(* CODESYS project Projeto_Silos.project

Project tree, tasks and I/O mapping:
  Device : CODESYS Control Win V3, 3S - Smart Software Solutions GmbH, order no. 305021, version 3.5.11.40
    application Application
      libraries: Standard, * (System)
      task Task_Simulacao (cyclic, interval t#20ms, priority 10) calls PRG_Simulacao
      task Task_Controle (cyclic, interval t#100ms, priority 5) calls PRG_Controle
      program PLC_PRG [ST]
      global variables GVL_IO
      global variables GVL_SCADA
      program PRG_Simulacao [ST]
      program PRG_Controle [SFC]: Enchimento, Acao_Parar_Tudo, Acao_Mover_SL01, Parar, Decisao_Alvo, Monitoramento_Falha, Comando_Atuadores, Adicionar_Peso, Remover_Peso
      Symbols
*)

// Device/Application/GVL_IO
VAR_GLOBAL
	
 
    (* ENTRADAS DO CLP (Sinais lidos e simulados pelo PRG_Simulacao) *)
   
    LS_01 : BOOL; (* Chave fim-de-curso Silo 1. TRUE quando Tripper posicionado. *)
    LS_02 : BOOL; (* Chave fim-de-curso Silo 2. *)
    LS_03 : BOOL; (* Chave fim-de-curso Silo 3. *)
    LS_04 : BOOL; (* Chave fim-de-curso Silo 4. *)
    
    TR_DIST : REAL; (* Sensor de distância a laser (metragem) . *)
    WT_01   : REAL; (* Balança de fluxo interna ao tripper (kg/s) . *)

 
    (* SAÍDAS DO CLP (Atuadores comandados pelo PRG_Controle) *)
  
    TR_FW   : BOOL; (* Acionamento frente do Tripper. *)
    TR_BW   : BOOL; (* Acionamento ré do Tripper. *)
    TR_VEL  : REAL; (* Velocidade de deslocamento do Tripper (m/s) . *)
    M_CT_01 : BOOL; (* Liga/desliga a correia alimentadora CT-01. *)
    BUZINA  : BOOL; (* Ativa a Buzina para sinalização. *)

END_VAR

// Device/Application/GVL_SCADA
VAR_GLOBAL
	
   
    (* COMANDOS/ENTRADAS LÓGICAS DO SCADA (Comandos para o CLP) *)

    LIGA_AUTO : BOOL; (* Comando de LIGA / DESLIGA executado via SCADA. *)
    EMG       : BOOL; (* Sinalização manual de Emergência via SCADA. *)
    REARME    : BOOL; (* Sinalização manual de Rearme via SCADA. *)
    
    FV_01     : BOOL; (* Válvula on-off de descarga Silo 1. *)
    FV_02     : BOOL; (* Válvula on-off de descarga Silo 2. *)
    FV_03     : BOOL; (* Válvula on-off de descarga Silo 3. *)
    FV_04     : BOOL; (* Válvula on-off de descarga Silo 4. *)
    
    LT_01     : REAL; (* Sensor de nível Silo 1 (Simulado manualmente via IHM, conforme orientação [cite: 123]). *)
    LT_02     : REAL; (* Sensor de nível Silo 2 (Simulado manualmente via IHM). *)
    LT_03     : REAL; (* Sensor de nível Silo 3 (Simulado manualmente via IHM). *)
    LT_04     : REAL; (* Sensor de nível Silo 4 (Simulado manualmente via IHM). *)

    
    (* DADOS/STATUS PARA VISUALIZAÇÃO NO SCADA (CLP envia para IHM) *)

    PESO_SL_01 : REAL; (* Peso total em toneladas do Silo 1[cite: 94]. *)
    PESO_SL_02 : REAL; (* Peso total em toneladas do Silo 2. *)
    PESO_SL_03 : REAL; (* Peso total em toneladas do Silo 3. *)
    PESO_SL_04 : REAL; (* Peso total em toneladas do Silo 4. *)
    
    STATUS_FALHA : BOOL; (* Indica que o CLP entrou em modo FALHA[cite: 64]. *)
    STATUS_EMG   : BOOL; (* Status da Emergência (para Alarme). *)
    POS_TRIPPER  : REAL; (* Posição atual do Tripper para Animação Visual. *)
    
    (* Variáveis para simulação de falha das chaves Fim-de-Curso via IHM [cite: 133] *)
    FALHA_LS_01 : BOOL;
    FALHA_LS_02 : BOOL;
    FALHA_LS_03 : BOOL;
    FALHA_LS_04 : BOOL;
	
	siloAlvo     : INT := 0; (* Silo alvo do tripper *)
	carregando   : BOOL;
	
END_VAR

// Device/Application/PRG_Simulacao
PROGRAM PRG_Simulacao
(* ==========================================================
 1. DECLARAÇÃO DE TODAS AS VARIÁVEIS
==========================================================
*)

(* Variáveis Temporárias *)
VAR
    fDeslocamentoCiclo : REAL;
END_VAR

(* Variáveis Constantes para posições *)
VAR CONSTANT
    fPosSilo_01 : REAL := 00.0; (* Posição central do Silo 1 em metros *)
    fPosSilo_02 : REAL := 10.0; (* Posição central do Silo 2 em metros *)
    fPosSilo_03 : REAL := 20.0; (* Posição central do Silo 3 em metros *)
    fPosSilo_04 : REAL := 30.0; (* Posição central do Silo 4 em metros *)
    fMargemPos  : REAL := 0.1;  (* Margem de 10cm para considerar "centro" *)
	fLimiteMaxPista : REAL := 30.0; (* A pista termina no silo 4 (30m)*)
END_VAR

(* ========================================================== 
 2. INÍCIO DA LÓGICA DO PROGRAMA 
==========================================================
*)

(* ==========================================================
 2.1 CÁLCULO DO DESLOCAMENTO DO TRIPPER (TR_DIST) 
==========================================================
*)
fDeslocamentoCiclo := TR_VEL * 0.02; (* Ciclo de 20ms = 0.02s *)

(* Atualiza a posição (TR_DIST) com base na direção *)
IF TR_FW AND (NOT TR_BW) THEN
    (* Movendo para frente *)
    TR_DIST := TR_DIST + fDeslocamentoCiclo;

ELSIF TR_BW AND (NOT TR_FW) THEN
    (* Movendo para trás *)
    TR_DIST := TR_DIST - fDeslocamentoCiclo;

ELSIF (TR_FW AND TR_BW) OR (NOT TR_FW AND NOT TR_BW) THEN
    (* Parado ou em condição de falha (ambos acionados) *)
    (* Não faz nada, a posição fica a mesma *)
END_IF;

(* Garante que a posição não fique negativa *)
IF TR_DIST < 0.0 THEN
    TR_DIST := 0.0;
END_IF;

(* ==========================================================
 2.2 SIMULAÇÃO DAS CHAVES FIM-DE-CURSO (LS_XX) 
==========================================================
*)

(* Silo 1 *)
IF (TR_DIST >= (fPosSilo_01 - fMargemPos)) AND 
   (TR_DIST <= (fPosSilo_01 + fMargemPos)) AND
   (NOT FALHA_LS_01) THEN 
    LS_01 := TRUE;
ELSE
    LS_01 := FALSE;
END_IF;

(* Silo 2 *)
IF (TR_DIST >= (fPosSilo_02 - fMargemPos)) AND 
   (TR_DIST <= (fPosSilo_02 + fMargemPos)) AND
   (NOT FALHA_LS_02) THEN
    LS_02 := TRUE;
ELSE
    LS_02 := FALSE;
END_IF;

(* Silo 3 *)
IF (TR_DIST >= (fPosSilo_03 - fMargemPos)) AND 
   (TR_DIST <= (fPosSilo_03 + fMargemPos)) AND
   (NOT FALHA_LS_03) THEN
    LS_03 := TRUE;
ELSE
    LS_03 := FALSE;
END_IF;

(* Silo 4 *)
IF (TR_DIST >= (fPosSilo_04 - fMargemPos)) AND 
   (TR_DIST <= (fPosSilo_04 + fMargemPos)) AND
   (NOT FALHA_LS_04) THEN
    LS_04 := TRUE;
ELSE
    LS_04 := FALSE;
END_IF;

(* ==========================================================
 2.3 SIMULAÇÃO DA BALANÇA DE FLUXO (WT_01) 
==========================================================
*)

IF M_CT_01 THEN 
    WT_01 := 1000.0; (* Vazão mássica constante de 1000 kg/s *)
ELSE
    WT_01 := 0.0;
END_IF;

(* Garante que a posição não exceda o limite máximo *)
IF TR_DIST > fLimiteMaxPista THEN
    TR_DIST := fLimiteMaxPista;
END_IF;

(* Garante que a posição não fique negativa *)
IF TR_DIST < 0.0 THEN
    TR_DIST := 0.0;
END_IF;

END_PROGRAM

// Device/Application/PRG_Controle
PROGRAM PRG_Controle
VAR

    PesoAdicionado_Ciclo : REAL;
    PesoRemovido_Ciclo   : REAL;
    TempoCiclo_s         : REAL := 0.1; (* 100ms *)

	Timer_Falha_Tripper   : TON; (* O bloco do temporizador *)
    bMovendo              : BOOL; (* Variável para saber se o tripper está se movendo *)
    bFalhaTimerTripper    : BOOL; (* A SAÍDA do timer (o alarme) *)
	(* --- Novas Variáveis de Estado da Lógica de Enchimento --- *)
    

    	
	posicaoAlvo     : REAL := 0.0; (* Posição (em metros) para onde o tripper deve ir *)
    distanciaAlvo   : REAL := 0.0; (* Distância restante até o alvo *)
    emPosicao       : BOOL := FALSE; (* TRUE se o tripper está no alvo (LS_XX) *)
	
	(* --- Variáveis para Lógica "Mais Próximo" --- *)
    distSilo1 : REAL;
    distSilo2 : REAL;
    distSilo3 : REAL;
    distSilo4 : REAL;
    distMinima : REAL;
	
	distanciaHome : REAL;
	
END_VAR


VAR CONSTANT
		(* --- Constantes de Nível (Capacidade 5000kg) --- *)
    Nivel_Baixo  : REAL := 500.0;  (* 10% da capacidade  *)
    Nivel_50pct  : REAL := 2500.0; (* 50%  *)
    Nivel_Alto   : REAL := 4500.0;  (* 90%  *)
	
	PosSilo_01 : REAL := 0.0; (* Posição central do Silo 1 em metros *)
    PosSilo_02 : REAL := 10.0; (* Posição central do Silo 2 em metros *)
    PosSilo_03 : REAL := 20.0; (* Posição central do Silo 3 em metros *)
    PosSilo_04 : REAL := 30.0; (* Posição central do Silo 4 em metros *)
	
END_VAR

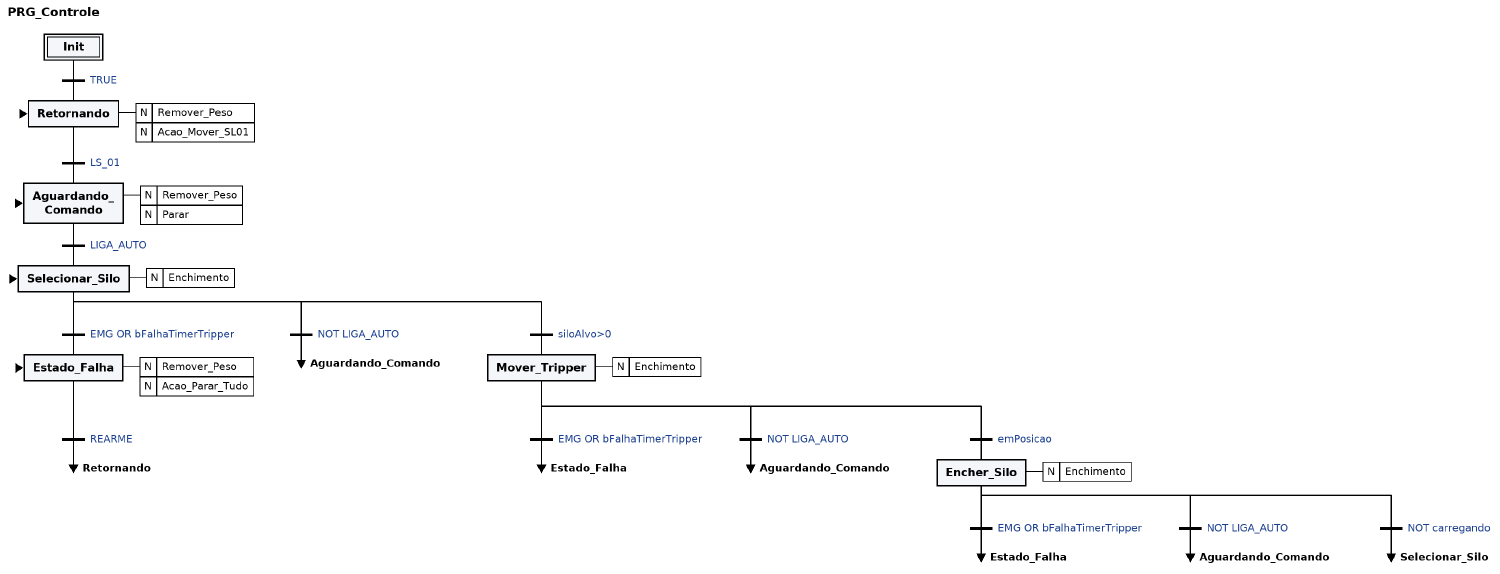
INITIAL_STEP Init:
END_STEP
TRANSITION FROM Init TO Retornando
    := TRUE;
END_TRANSITION
STEP Retornando:
    Remover_Peso(N);
    Acao_Mover_SL01(N);
END_STEP
TRANSITION FROM Retornando TO Aguardando_Comando
    := LS_01;
END_TRANSITION
STEP Aguardando_Comando:
    Remover_Peso(N);
    Parar(N);
END_STEP
TRANSITION FROM Aguardando_Comando TO Selecionar_Silo
    := LIGA_AUTO;
END_TRANSITION
STEP Selecionar_Silo:
    Enchimento(N);
END_STEP
TRANSITION FROM Selecionar_Silo TO Estado_Falha
    := EMG OR bFalhaTimerTripper;
END_TRANSITION
STEP Estado_Falha:
    Remover_Peso(N);
    Acao_Parar_Tudo(N);
END_STEP
TRANSITION FROM Estado_Falha TO Retornando
    := REARME;
END_TRANSITION
TRANSITION FROM Selecionar_Silo TO Aguardando_Comando
    := NOT LIGA_AUTO;
END_TRANSITION
TRANSITION FROM Selecionar_Silo TO Mover_Tripper
    := siloAlvo>0;
END_TRANSITION
STEP Mover_Tripper:
    Enchimento(N);
END_STEP
TRANSITION FROM Mover_Tripper TO Estado_Falha
    := EMG OR bFalhaTimerTripper;
END_TRANSITION
TRANSITION FROM Mover_Tripper TO Aguardando_Comando
    := NOT LIGA_AUTO;
END_TRANSITION
TRANSITION FROM Mover_Tripper TO Encher_Silo
    := emPosicao;
END_TRANSITION
STEP Encher_Silo:
    Enchimento(N);
END_STEP
TRANSITION FROM Encher_Silo TO Estado_Falha
    := EMG OR bFalhaTimerTripper;
END_TRANSITION
TRANSITION FROM Encher_Silo TO Aguardando_Comando
    := NOT LIGA_AUTO;
END_TRANSITION
TRANSITION FROM Encher_Silo TO Selecionar_Silo
    := NOT carregando;
END_TRANSITION

ACTION Enchimento:
(* Esta ação agrupa TODAS as lógicas enquanto o sistema está RODANDO *)

(* 1. Matemáticas de Peso *)
Adicionar_Peso();  (* Calcula entrada no silo *)
Remover_Peso();    (* Calcula saída do silo *)

(* 2. Controle e Segurança *)
Monitoramento_Falha();  (* Verifica timer de 5s *)
Decisao_Alvo();         (* Define quem encher e quando parar *)
Comando_Atuadores();    (* Move o tripper e liga a esteira *)
END_ACTION

ACTION Acao_Parar_Tudo:
(* Ação ST executada continuamente em Estado_Falha *)
TR_VEL := 0.0;
TR_FW := FALSE;
TR_BW := FALSE;
M_CT_01 := FALSE;
BUZINA := TRUE; (* Liga a buzina de alarme *)

(* 2. Reset de Comandos (CORREÇÃO) *)
LIGA_AUTO := FALSE; (* Força o botão Automático a desligar *)

(* 3. Reset Lógico *)
carregando := FALSE;
siloAlvo := 0;
posicaoAlvo := TR_DIST;
END_ACTION

ACTION Acao_Mover_SL01:
(* ============================================ *)
(* Ação ST executada continuamente em "Retornando" *)
(* ============================================ *)

(*
Esta lógica move o tripper para a Posição "Home" (PosSilo_01 = 0.0m)
usando a tabela de desaceleração.
*)

(*Resets*)

EMG := FALSE;       (* Destrava a Emergência *)
LIGA_AUTO := FALSE; (* Garante que não parta sozinho *)
STATUS_FALHA := FALSE; (* Apaga o alarme de falha se houver *)
siloAlvo := 1;

(* Calcula a distância restante até o Silo 1 *)
distanciaHome := ABS(PosSilo_01 - TR_DIST);

(* Verifica se já chegou *)
IF LS_01 OR (distanciaHome < 0.1) THEN
    (* Chegou no SL-01 *)
    TR_VEL := 0.0;
    TR_FW := FALSE;
    TR_BW := FALSE;
	siloAlvo := 0;
ELSE
    (* Ainda não chegou, aplicar desaceleração *)
    IF distanciaHome > 30.0 THEN
        TR_VEL := 5.0;
    ELSIF distanciaHome > 25.0 THEN
        TR_VEL := 4.5;
    ELSIF distanciaHome > 20.0 THEN
        TR_VEL := 4.0;
    ELSIF distanciaHome > 15.0 THEN
        TR_VEL := 2.5;
    ELSIF distanciaHome > 10.0 THEN
        TR_VEL := 1.5;
    ELSIF distanciaHome > 5.0 THEN
        TR_VEL := 1;
    ELSE
        TR_VEL := 0.5;
    END_IF;

    (* Definir Direção (assumindo SL-01 está na posição 10.0) *)
    IF PosSilo_01 < TR_DIST THEN
        (* Tripper está à frente (ex: 20m), precisa ir para trás *)
        TR_FW := FALSE;
        TR_BW := TRUE;
    ELSE
        (* Tripper está atrás (ex: 5m), precisa ir para frente *)
        TR_FW := TRUE;
        TR_BW := FALSE;
    END_IF;
END_IF;
END_ACTION

ACTION Parar:
(* ============================================ *)
(* Ação para garantir que todos os atuadores de movimento estejam desligados *)
(* ============================================ *)

TR_VEL := 0.0;
TR_FW := FALSE;
TR_BW := FALSE;
M_CT_01 := FALSE;
END_ACTION

ACTION Decisao_Alvo:
(* ============================================ *)
(* 5. LÓGICA DE CONTROLE DE ENCHIMENTO (REFINADA) *)
(* ============================================ *)

(* --- Regra: Carregamento não pode ser interrompido --- *)
IF carregando THEN
    (* ESTADO 1: JÁ ESTAMOS CARREGANDO UM SILO *)
    
    (* Lógica de Parada: O silo alvo atingiu o Nível Alto? *)
    IF (siloAlvo = 1 AND PESO_SL_01 >= Nivel_Alto) OR
       (siloAlvo = 2 AND PESO_SL_02 >= Nivel_Alto) OR
       (siloAlvo = 3 AND PESO_SL_03 >= Nivel_Alto) OR
       (siloAlvo = 4 AND PESO_SL_04 >= Nivel_Alto) THEN
        
        (* SIM: Parar o carregamento e resetar o estado *)
        carregando := FALSE;
        siloAlvo := 0;
        (* Nota: O desligamento da correia M_CT_01 é feito na ação Comando_Atuadores *)
    END_IF;

ELSE
    (* ESTADO 2: NÃO ESTAMOS CARREGANDO - SELECIONAR NOVO ALVO *)
    
    siloAlvo := 0; (* Reseta o alvo *)
    distMinima := 1000.0; (* Valor alto para iniciar a comparação *)

    (* --- Cálculo das distâncias atuais --- *)
    distSilo1 := ABS(TR_DIST - PosSilo_01);
    distSilo2 := ABS(TR_DIST - PosSilo_02);
    distSilo3 := ABS(TR_DIST - PosSilo_03);
    distSilo4 := ABS(TR_DIST - PosSilo_04);

    (* --- Lógica de Prioridade 1: Nível Baixo (< 10%) --- *)
    IF PESO_SL_01 < Nivel_Baixo THEN
        distMinima := distSilo1;
        siloAlvo := 1;
    END_IF;
    IF PESO_SL_02 < Nivel_Baixo AND distSilo2 < distMinima THEN
        distMinima := distSilo2;
        siloAlvo := 2;
    END_IF;
    IF PESO_SL_03 < Nivel_Baixo AND distSilo3 < distMinima THEN
        distMinima := distSilo3;
        siloAlvo := 3;
    END_IF;
    IF PESO_SL_04 < Nivel_Baixo AND distSilo4 < distMinima THEN
        distMinima := distSilo4;
        siloAlvo := 4;
    END_IF;

    (* --- Lógica de Prioridade 2: Nível < 50% --- *)
    (* Só executa se NENHUM silo foi selecionado pela Prioridade 1 *)
    IF siloAlvo = 0 THEN
        IF PESO_SL_01 < Nivel_50pct THEN siloAlvo := 1;
        ELSIF PESO_SL_02 < Nivel_50pct THEN siloAlvo := 2;
        ELSIF PESO_SL_03 < Nivel_50pct THEN siloAlvo := 3;
        ELSIF PESO_SL_04 < Nivel_50pct THEN siloAlvo := 4;
        END_IF;
    END_IF;
    
    (* Se encontramos um alvo, iniciamos o processo *)
    IF siloAlvo > 0 THEN
        carregando := TRUE;
    END_IF;
END_IF;
END_ACTION

ACTION Monitoramento_Falha:
(* ============================================ *)
(* 4. LÓGICA DE DETECÇÃO DE FALHA (5 SEGUNDOS) *)
(* ============================================ *)

(*
A condição de falha (IN) é:
1. O sistema está tentando carregar (carregando = TRUE)
2. E o motor do tripper parou (TR_VEL = 0.0)
3. Mas a chave fim-de-curso NÃO foi atuada (emPosicao = FALSE)
*)

Timer_Falha_Tripper(
    IN:= carregando AND (TR_VEL = 0.0) AND (NOT emPosicao) AND (siloAlvo > 0),
    PT:= T#5S,
    Q=> bFalhaTimerTripper (* Saída booleana que usamos na transição SFC *)
);
STATUS_FALHA := bFalhaTimerTripper;
END_ACTION

ACTION Comando_Atuadores:
(* ============================================ *)
(* 6. LÓGICA DE MOVIMENTO E COMANDO DE ATUADORES *)
(* ============================================ *)

(* --- Parte A: Definir para onde ir (Posição Alvo) --- *)
IF siloAlvo = 1 THEN posicaoAlvo := PosSilo_01;
ELSIF siloAlvo = 2 THEN posicaoAlvo := PosSilo_02;
ELSIF siloAlvo = 3 THEN posicaoAlvo := PosSilo_03;
ELSIF siloAlvo = 4 THEN posicaoAlvo := PosSilo_04;
ELSE posicaoAlvo := TR_DIST; (* Ficar onde está *)
END_IF;

(* --- Parte B: Calcular distância e verificar posição --- *)
distanciaAlvo := ABS(posicaoAlvo - TR_DIST); (* Distância absoluta *)
emPosicao := (LS_01 AND siloAlvo = 1) OR 
             (LS_02 AND siloAlvo = 2) OR 
             (LS_03 AND siloAlvo = 3) OR
             (LS_04 AND siloAlvo = 4);

(* --- Parte C: Lógica de Movimento e Desaceleração --- *)
IF carregando AND NOT emPosicao THEN
    (* MOVER: Aplicar Tabela de Desaceleração *)
    IF distanciaAlvo > 30.0 THEN TR_VEL := 5.0;
    ELSIF distanciaAlvo > 25.0 THEN TR_VEL := 4.5;
    ELSIF distanciaAlvo > 20.0 THEN TR_VEL := 4.0;
    ELSIF distanciaAlvo > 15.0 THEN TR_VEL := 2.5;
    ELSIF distanciaAlvo > 10.0 THEN TR_VEL := 1.5;
    ELSIF distanciaAlvo > 5.0 THEN TR_VEL := 1.0;
    ELSIF distanciaAlvo > 0.1 THEN TR_VEL := 0.5;
    ELSE TR_VEL := 0.0;
    END_IF;
    
    (* Definir Direção *)
    IF posicaoAlvo > TR_DIST THEN
        TR_FW := TRUE; TR_BW := FALSE;
    ELSIF posicaoAlvo < TR_DIST THEN
        TR_FW := FALSE; TR_BW := TRUE;
    END_IF;
    
    M_CT_01 := FALSE; (* Correia desligada durante movimento *)

ELSIF carregando AND emPosicao THEN
    (* CARREGAR: Parar e Ligar Correia *)
    TR_VEL := 0.0;
    TR_FW := FALSE;
    TR_BW := FALSE;
    M_CT_01 := TRUE; (* LIGA A CORREIA *)

ELSE
    (* PARADO: Desligar tudo *)
    TR_VEL := 0.0;
    TR_FW := FALSE;
    TR_BW := FALSE;
    M_CT_01 := FALSE;
END_IF;
END_ACTION

ACTION Adicionar_Peso:

(*  CÁLCULO DO PESO CARREGADO (ENCHIMENTO) *)

(* WT_01 informa kg/s. O ciclo é 0,1s *)
PesoAdicionado_Ciclo := WT_01 * TempoCiclo_s;

(* Só adiciona peso se a correia (M_CT_01) estiver ligada
   E o tripper estiver sobre o silo correto (LS_XX) *)

IF M_CT_01 AND LS_01 THEN
    PESO_SL_01 := PESO_SL_01 + PesoAdicionado_Ciclo;
ELSIF M_CT_01 AND LS_02 THEN
    PESO_SL_02 := PESO_SL_02 + PesoAdicionado_Ciclo;
ELSIF M_CT_01 AND LS_03 THEN
    PESO_SL_03 := PESO_SL_03 + PesoAdicionado_Ciclo;
ELSIF M_CT_01 AND LS_04 THEN
    PESO_SL_04 := PESO_SL_04 + PesoAdicionado_Ciclo;
END_IF;

(* GARANTIR LIMITES DE PESO *)

IF PESO_SL_01 < 0.0 THEN PESO_SL_01 := 0.0; END_IF;
IF PESO_SL_01 > 5000.0 THEN PESO_SL_01 := 5000.0; END_IF;

IF PESO_SL_02 < 0.0 THEN PESO_SL_02 := 0.0; END_IF;
IF PESO_SL_02 > 5000.0 THEN PESO_SL_02 := 5000.0; END_IF;

IF PESO_SL_03 < 0.0 THEN PESO_SL_03 := 0.0; END_IF;
IF PESO_SL_03 > 5000.0 THEN PESO_SL_03 := 5000.0; END_IF;

IF PESO_SL_04 < 0.0 THEN PESO_SL_04 := 0.0; END_IF;
IF PESO_SL_04 > 5000.0 THEN PESO_SL_04 := 5000.0; END_IF;
END_ACTION

ACTION Remover_Peso:
(* CÁLCULO DO PESO VAZADO (ESVAZIAMENTO) *)

(* O operador pode esvaziar a qualquer momento *)

PesoRemovido_Ciclo := 500.0 * TempoCiclo_s; (* 500 kg/s * 0.1s = 50 kg *)

IF FV_01 THEN
    PESO_SL_01 := PESO_SL_01 - PesoRemovido_Ciclo;
END_IF;
IF FV_02 THEN
    PESO_SL_02 := PESO_SL_02 - PesoRemovido_Ciclo;
END_IF;
IF FV_03 THEN
    PESO_SL_03 := PESO_SL_03 - PesoRemovido_Ciclo;
END_IF;
IF FV_04 THEN
    PESO_SL_04 := PESO_SL_04 - PesoRemovido_Ciclo;
END_IF;


(* GARANTIR LIMITES DE PESO *)

IF PESO_SL_01 < 0.0 THEN PESO_SL_01 := 0.0; END_IF;
IF PESO_SL_01 > 5000.0 THEN PESO_SL_01 := 5000.0; END_IF;

IF PESO_SL_02 < 0.0 THEN PESO_SL_02 := 0.0; END_IF;
IF PESO_SL_02 > 5000.0 THEN PESO_SL_02 := 5000.0; END_IF;

IF PESO_SL_03 < 0.0 THEN PESO_SL_03 := 0.0; END_IF;
IF PESO_SL_03 > 5000.0 THEN PESO_SL_03 := 5000.0; END_IF;

IF PESO_SL_04 < 0.0 THEN PESO_SL_04 := 0.0; END_IF;
IF PESO_SL_04 > 5000.0 THEN PESO_SL_04 := 5000.0; END_IF;
END_ACTION

END_PROGRAM

// Device/Application/PLC_PRG
PROGRAM PLC_PRG
VAR
END_VAR

END_PROGRAM
